Universal Robots PolyScope program: Putback_program.urp

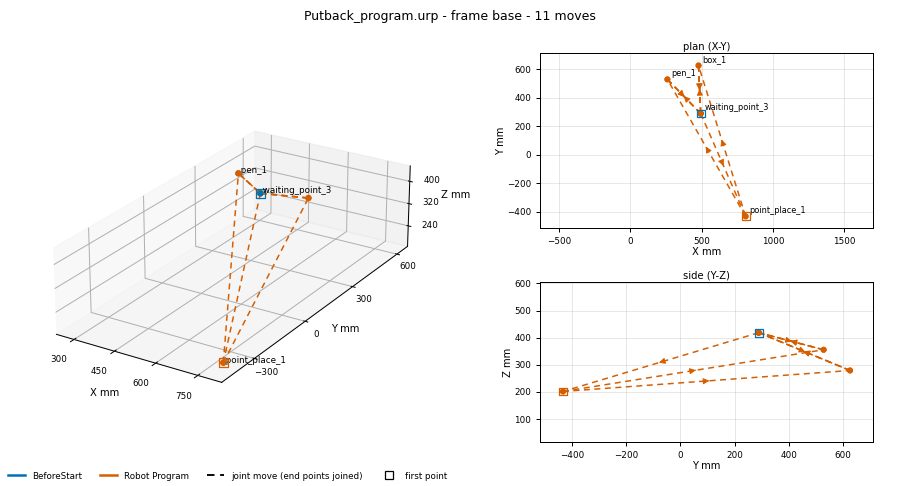
[picture p0: tool path of Putback_program.urp in frame base, 11 of 11 moves have a stored position in this frame; points joined in program order, loops and branches not executed]
Program Putback_program (installation=default directory=/ursim/programs/MQTT createdIn=5.16.0 lastSavedIn=5.16.0 robotSerialNumber=20195599999)
Calibrated DH parameters: a=[0, -0.425, -0.3922, 0, 0, 0]; d=[0.1625, 0, 0, 0.1333, 0.0997, 0.0996]; alpha=[1.570796, 0, 0, 1.570796, -1.570796, 0]; deltaTheta=[0, 0, 0, 0, 0, 0]
InitVariablesNode variables(variable(name=cmd_name, expression=" "), variable(name=object, expression=" "), variable(name=object_hold, expression=" "), variable(name=params, expression=" "), variable(name=topic_order, expression="robot/order"))
BeforeStart
  Script file /ursim/programs/MQTT/json.script
    | ###
    | # summary: This function is used to split a string into an array of substrings with a delimiter
    | # @param str :string the string to split
    | # @param delimiter :string the caracter to split the string
    | # @param debug :bool activ message debug
    | ###
    | MAX_VARIABLES = 100
    | def str_split(str, delimiter, debug=False):
    |   result = make_list(0, "", MAX_VARIABLES) # Arrays to stock the result max 10 variables
    |   start = 0  # Position to start the search
    |   end_deli = str_find(str, delimiter) #Find the first delimiter
    | 
    |   # While a delimiter is found
    |   while end_deli != -1:
    |     if result.excess_capacity() == 0:
    |       if debug:
    |         textmsg("Number of variables exceeded")
    |       end
    |       return result
    |     end
    | 
    |     # Extraction of the substring between the start and the delimiter
    |     substring = str_sub(str, start, end_deli - start)
    |     result.append(substring)
    | 
    |     # Update the start position and the end delimiter
    |     str = str_sub(str, end_deli + str_len(delimiter), str_len(str))
    |     end_deli = str_find(str, delimiter)
    |   end
    | 
    |   # Add the last substring
    |   if result.excess_capacity() > 0:
    |     result.append(str)
    |   elif debug:
    |     textmsg("Number of variables exceeded")
    |   end
    | 
    |   if debug:
    |     textmsg("Result: " + result.to_string())
    |   end
    |   return result
    | end
    | 
    | 
    | ###
    | # summary: This function to return the value of a variable in a JSON string function only with string type
    | # @param json_string :string the json payload
    | # @param variable :string the variable the function needs to find
    | # @param debug :bool activ message debug
    | ###
    | def value_json_string(json_string, variable, type="str",debug=False):
    |   #Verify the json string is not empty (2 brackets at minimal)
    |   if str_len(json_string) < 2:
    |     if debug:
    |       textmsg("The JSON string is empty or invalid")
    |     end
    |     if(type == "int"):
    |       return 0
    |     end
    |     return " "
    |   end
    | 
    |   json_string = str_sub(json_string, 1, str_len(json_string) - 2) #Cut the first and last bracket
    |   variable_array = str_split(json_string, ",", debug) #Split the json string into an array of variables
    | 
    |   idx = 0 #Index of the array
    |   len_var_array = variable_array.length() #Length of the array
    | 
    |   #While the index is less than the length of the array
    |   while idx < len_var_array:
    | 
    |     find = str_find(variable_array[idx], variable) #Find the variable in the array
    |     if find > 0: #If the variable is found
    |       if debug:
    |         textmsg("Variable found")
    |       end
    |       value = str_split(variable_array[idx], ":")[1] #Split the variable to get the value
    |       if str_find(value, "'")>0: #If the value is a string
    |         return str_sub(value, 2, str_len(value) - 3) #Return the value without the quotes
    |       end
    |       if(type == "int"):
    |         return to_num(value)
    |       end
    |       return str_sub(value, 1, str_len(value) - 2) #Return the value without the quotes
    |     end
    |     idx = idx + 1
    |   end
    |   if(type == "int"):
    |     return 0
    |   end
    |   return " "
    | end
  params := "{'object':'pen'}"
  object_hold := ""
  MoveJ speed 60 deg/s, acceleration 80 deg/s^2 (useActiveTCP=true) feature=Base
    Waypoint waiting_point_3: TCP in base x=492.803 y=288.649 z=418.324 mm, rx=2.6568 ry=-1.6608 rz=-0.0199 rad; joints [192.415, -98.238, 124.325, -115.253, -89.954, -13.481] deg
Robot Program (runOnlyOnce=true)
  object := value_json_string(params, "object")
  If object == "pen" and object_hold == " "
    Folder take object
      MoveJ speed 60 deg/s, acceleration 80 deg/s^2 (useActiveTCP=true) feature=Base
        Waypoint point_place_1: TCP in base x=807.912 y=-433.125 z=201.587 mm, rx=-0.6852 ry=3.024 rz=-0.0161 rad; joints [140.573, -55.8, 96.757, -132.886, -88.708, 25.083] deg
      MoveL speed 250 mm/s, acceleration 1200 mm/s^2 (useActiveTCP=true) feature=Joint_6_name
        MoveDirectionNode (selectedDirection=ZPlus)
          Until DISTANCE (allowActions=false deceleration=3 distanceNodeType=STOP) Distance=0.05; motionParameters(blendRadius=0)
          Until TOOL_CONTACT_DETECTION (allowActions=false retraction=0.002 decelerationAcceleration=3 decelerationAngularAcceleration=34.906585)
        MoveDirectionNode (selectedDirection=ZMinus) feature=Joint_6_name
          Until DISTANCE (allowActions=false deceleration=3 distanceNodeType=STOP) Distance=0.05; motionParameters(blendRadius=0)
    Folder put back
      MoveJ speed 60 deg/s, acceleration 80 deg/s^2 (useActiveTCP=true) feature=Base
        Waypoint pen_1: TCP in base x=259.212 y=527.898 z=355.358 mm, rx=-2.6848 ry=1.6264 rz=-0.0183 rad; joints [226.614, -92.85, 127.172, -124.624, -90.757, 19.087] deg
      MoveL speed 250 mm/s, acceleration 1200 mm/s^2 (useActiveTCP=true) feature=Base
        MoveDirectionNode (selectedDirection=ZMinus toolParams=0.05, 1.2) feature=Base
          Until DISTANCE (allowActions=false deceleration=3 distanceNodeType=STOP) Distance=0.05; motionParameters(blendRadius=0)
          Until TOOL_CONTACT_DETECTION (allowActions=false retraction=0.003 decelerationAcceleration=3 decelerationAngularAcceleration=34.906585)
        MoveDirectionNode (selectedDirection=ZPlus)
          Until DISTANCE (allowActions=false deceleration=3 distanceNodeType=STOP) Distance=0.005; motionParameters(blendRadius=0)
    MoveJ speed 60 deg/s, acceleration 80 deg/s^2 (useActiveTCP=true) feature=Base
      Waypoint waiting_point_4: TCP in base x=492.803 y=288.649 z=418.324 mm, rx=2.6568 ry=-1.6608 rz=-0.0199 rad; joints [192.415, -98.238, 124.325, -115.253, -89.954, -13.481] deg
    object_hold := " "
  ElseIf object == "box" and object_hold == " "
    Folder take object
      MoveJ speed 60 deg/s, acceleration 80 deg/s^2 (useActiveTCP=true) feature=Base
        Waypoint point_place_2: TCP in base x=807.912 y=-433.125 z=201.587 mm, rx=-0.6852 ry=3.024 rz=-0.0161 rad; joints [140.573, -55.8, 96.757, -132.886, -88.708, 25.083] deg
      MoveL speed 250 mm/s, acceleration 1200 mm/s^2 (useActiveTCP=true) feature=Joint_6_name
        MoveDirectionNode (selectedDirection=ZPlus)
          Until DISTANCE (allowActions=false deceleration=3 distanceNodeType=STOP) Distance=0.05; motionParameters(blendRadius=0)
          Until TOOL_CONTACT_DETECTION (allowActions=false retraction=0.002 decelerationAcceleration=3 decelerationAngularAcceleration=34.906585)
        MoveDirectionNode (selectedDirection=ZMinus) feature=Joint_6_name
          Until DISTANCE (allowActions=false deceleration=3 distanceNodeType=STOP) Distance=0.05; motionParameters(blendRadius=0)
    Folder put back
      MoveJ speed 60 deg/s, acceleration 80 deg/s^2 (useActiveTCP=true) feature=Base
        Waypoint box_1: TCP in base x=477.624 y=625.24 z=278.948 mm, rx=-2.6325 ry=1.6869 rz=0.0449 rad; joints [219.454, -70.395, 109.973, -129.892, -88.344, 14.805] deg
      MoveL speed 250 mm/s, acceleration 1200 mm/s^2 (useActiveTCP=true) feature=Base
        MoveDirectionNode (selectedDirection=ZMinus toolParams=0.05, 1.2) feature=Base
          Until DISTANCE (allowActions=false deceleration=3 distanceNodeType=STOP) Distance=0.05; motionParameters(blendRadius=0)
          Until TOOL_CONTACT_DETECTION (allowActions=false retraction=0.003 decelerationAcceleration=3 decelerationAngularAcceleration=34.906585)
        MoveDirectionNode (selectedDirection=ZPlus)
          Until DISTANCE (allowActions=false deceleration=3 distanceNodeType=STOP) Distance=0.005; motionParameters(blendRadius=0)
    MoveJ speed 60 deg/s, acceleration 80 deg/s^2 (useActiveTCP=true) feature=Base
      Waypoint waiting_point_5: TCP in base x=492.803 y=288.649 z=418.324 mm, rx=2.6568 ry=-1.6608 rz=-0.0199 rad; joints [192.415, -98.238, 124.325, -115.253, -89.954, -13.481] deg
    object_hold := " "
  ElseIf object=="pen" and object_hold=="pen"
    Folder put back
      MoveJ speed 60 deg/s, acceleration 80 deg/s^2 (useActiveTCP=true) feature=Base
        Waypoint pen_1: TCP in base x=259.212 y=527.898 z=355.358 mm, rx=-2.6848 ry=1.6264 rz=-0.0183 rad; joints [226.614, -92.85, 127.172, -124.624, -90.757, 19.087] deg
      MoveL speed 250 mm/s, acceleration 1200 mm/s^2 (useActiveTCP=true) feature=Base
        MoveDirectionNode (selectedDirection=ZMinus toolParams=0.05, 1.2) feature=Base
          Until DISTANCE (allowActions=false deceleration=3 distanceNodeType=STOP) Distance=0.05; motionParameters(blendRadius=0)
          Until TOOL_CONTACT_DETECTION (allowActions=false retraction=0.003 decelerationAcceleration=3 decelerationAngularAcceleration=34.906585)
        MoveDirectionNode (selectedDirection=ZPlus)
          Until DISTANCE (allowActions=false deceleration=3 distanceNodeType=STOP) Distance=0.005; motionParameters(blendRadius=0)
    MoveJ speed 60 deg/s, acceleration 80 deg/s^2 (useActiveTCP=true) feature=Base
      Waypoint waiting_point_3: TCP in base x=492.803 y=288.649 z=418.324 mm, rx=2.6568 ry=-1.6608 rz=-0.0199 rad; joints [192.415, -98.238, 124.325, -115.253, -89.954, -13.481] deg
  ElseIf object=="box" and object_hold=="box"
    Folder put back
      MoveJ speed 60 deg/s, acceleration 80 deg/s^2 (useActiveTCP=true) feature=Base
        Waypoint box_1: TCP in base x=477.624 y=625.24 z=278.948 mm, rx=-2.6325 ry=1.6869 rz=0.0449 rad; joints [219.454, -70.395, 109.973, -129.892, -88.344, 14.805] deg
      MoveL speed 250 mm/s, acceleration 1200 mm/s^2 (useActiveTCP=true) feature=Base
        MoveDirectionNode (selectedDirection=ZMinus toolParams=0.05, 1.2) feature=Base
          Until DISTANCE (allowActions=false deceleration=3 distanceNodeType=STOP) Distance=0.05; motionParameters(blendRadius=0)
          Until TOOL_CONTACT_DETECTION (allowActions=false retraction=0.003 decelerationAcceleration=3 decelerationAngularAcceleration=34.906585)
        MoveDirectionNode (selectedDirection=ZPlus)
          Until DISTANCE (allowActions=false deceleration=3 distanceNodeType=STOP) Distance=0.005; motionParameters(blendRadius=0)
    MoveJ speed 60 deg/s, acceleration 80 deg/s^2 (useActiveTCP=true) feature=Base
      Waypoint waiting_point_4: TCP in base x=492.803 y=288.649 z=418.324 mm, rx=2.6568 ry=-1.6608 rz=-0.0199 rad; joints [192.415, -98.238, 124.325, -115.253, -89.954, -13.481] deg
  object_hold := " "
